// TIA Portal V17 program export: 0 tag tables, 0 data types, 1 data blocks, 2 code blocks (in call order from the OBs), 1 instance data blocks

DATA_BLOCK "Data_block_1"   // DB73
{ S7_Optimized_Access := 'TRUE' }
// stored: MemoryReserve 100
BEGIN
END_DATA_BLOCK

ORGANIZATION_BLOCK "Main"   // OB1, LAD, ProgramCycle
TITLE = "Main Program Sweep (Cycle)"
{ S7_Optimized_Access := 'TRUE' }
// stored: SetENOAutomatically false
   VAR_INPUT
      Initial_Call : Bool;   // Initial call of this OB
      Remanence : Bool;   // =True, if remanent data are available
   END_VAR
BEGIN
END_ORGANIZATION_BLOCK

FUNCTION_BLOCK "Main_Safety_RTG1"   // FB1, F_FBD
{ S7_Optimized_Access := 'TRUE' }
// stored: AutoNumber false
BEGIN
END_FUNCTION_BLOCK

DATA_BLOCK "Main_Safety_RTG1_DB"   // DB1, F_DB
NAME : FUSI
// stored: InstanceOfName Main_Safety_RTG1, InstanceOfType FB
"Main_Safety_RTG1"
BEGIN
END_DATA_BLOCK
